(* CoDeSys 2.3.9.62 project: MM000-P9000-00-A.pro *)
(* Author: JvL *)
(* Libraries: ifm_RAWCan\ifm_RAWCan_NT_V020004.lib 1.10.19 08:10:40, ifm_CR0403\ifm_CR0403_V030100.lib 22.3.17 12:39:40, ifm_CANopen\ifm_NetVarLib_NT_V020004.lib 1.10.19 08:10:40, standard.lib 4.10.05 12:14:46, SysLibCallback.lib 26.9.08 18:43:52, 3S_CANOPENNETVAR.LIB 23.10.20 12:28:45, Iecsfc.lib 2.6.14 11:37:46, Util.lib 23.10.20 12:25:49, ifm_CANopen\3S_CANopenManager.lib 23.10.20 12:28:45, ifm_CANopen\3S_CanDrv.lib 23.10.20 12:28:45 *)

(* PLC configuration (modules and I/O channels)
Configuration [LocalConfiguration] node 0, in %IB0 out %QB0 {IFM_PARAM_WORD_TIME = 0}
Inputs Binary [LocalIn] node 0, in %IB0 out %QB0
  IN00 AT %IB0 [ChInputBool] Input 00 Bit
  IN01 AT %IB1 [ChInputBool] Input 01 Bit
  IN02 AT %IB2 [ChInputBool] Input 02 Bit
  IN03 AT %IB3 [ChInputBool] Input 03 Bit
  IN04 AT %IB4 [ChInputBool] Input 04 Bit
  IN05 AT %IB5 [ChInputBool] Input 05 Bit
  IN06 AT %IB6 [ChInputBool] Input 06 Bit
  IN07 AT %IB7 [ChInputBool] Input 07 Bit
  IN08 AT %IB8 [ChInputBool] Input 08 Bit
  IN09 AT %IB9 [ChInputBool] Input 09 Bit
  IN10 AT %IB10 [ChInputBool] Input 10 Bit
  IN11 AT %IB11 [ChInputBool] Input 11 Bit
Outputs Binary [LocalOut] node 1, in %IB12 out %QB0
  OUT00 AT %QB0 [ChOutputBool] Output 00 Bit
  OUT01 AT %QB1 [ChOutputBool] Output 01 Bit
  OUT02 AT %QB2 [ChOutputBool] Output 02 Bit
  OUT03 AT %QB3 [ChOutputBool] Output 03 Bit
  OUT04 AT %QB4 [ChOutputBool] Output 04 Bit
  OUT05 AT %QB5 [ChOutputBool] Output 05 Bit
  OUT06 AT %QB6 [ChOutputBool] Output 06 Bit
  OUT07 AT %QB7 [ChOutputBool] Output 07 Bit
  OUT08 AT %QB8 [ChOutputBool] Output 08 Bit
  OUT09 AT %QB9 [ChOutputBool] Output 09 Bit
  OUT10 AT %QB10 [ChOutputBool] Output 10 Bit
  OUT11 AT %QB11 [ChOutputBool] Output 11 Bit
SUPPLY_VOLTAGE_VBBS AT %IW6 [ChInputWord] Supply voltage VBBS
SUPPLY_VOLTAGE_VU AT %IW7 [ChInputWord] Supply voltage VU
SUPPLY_VOLTAGE_VBB1 AT %IW8 [ChInputWord] Supply voltage VBB1
SUPPLY_VOLTAGE_VBB2 AT %IW9 [ChInputWord] Supply voltage VBB2
TEMPERATURE AT %IW10 [ChInputInt] Temperature
CAN Communication [LocalCANCom] node 2, in %IB22 out %QB12
  Interface CAN 1 [CAN_BUS] node 0, in %IB22 out %QB12 {STACK_DWORD_S = 0}
    CANopen Interface [CAN_OPEN] node 0, in %IB22 out %QB12
    J1939 Interface [CAN_J1939] node 1, in %IB22 out %QB12
  Interface CAN 2 [CAN_BUS] node 1, in %IB22 out %QB12 {STACK_DWORD_S = 0}
    CANopen Interface [CAN_OPEN] node 0, in %IB22 out %QB12
    J1939 Interface [CAN_J1939] node 1, in %IB22 out %QB12
*)

(* Global variable list: CanOpen implicit Variables *)
VAR_GLOBAL CONSTANT
	MAX_CTRLINDEX : INT := -1;
END_VAR

(* Global variable list: Global_Variables *)
VAR_GLOBAL
	encoderStatic:BOOL;
END_VAR

(* Global variable list: Networkmanagement implicit Variables CAN *)
VAR_GLOBAL CONSTANT
	USE_NWVARS_CAN : BOOL := TRUE;
	MAX_NetVarItems_CAN	: INT := 31;
	MAX_NetVarPDO_Rx_CAN	: INT := 3;
	MAX_NetVarPDO_Tx_CAN	: INT := 7;
	MAX_NetVarOD_CAN		: INT := 0;
END_VAR
VAR_GLOBAL
	pNetVarItems_CAN		: ARRAY[0..MAX_NetVarItems_CAN] OF NetVarDataItem_CAN;
	pNetVarPDO_Rx_CAN		: ARRAY[0..MAX_NetVarPDO_Rx_CAN] OF NetVarPDO_Rx_CAN;
	pNetVarPDO_Tx_CAN		: ARRAY[0..MAX_NetVarPDO_Tx_CAN] OF NetVarPDO_Tx_CAN;
	pNetVarOD_CAN			: ARRAY[0..MAX_NetVarOD_CAN] OF NetVarOD_CAN;
END_VAR

(* Global variable list: PDM_PLC_COMUNICATION2 *)
VAR_GLOBAL

	(*
	 System variables for basic comunication. CANopen TX/RX PDO1, PDO2, PDO3 and PDO4
	or CANLayer2 TX/RX COB1, COB2, COB3 and COB4
	*)


(************************************From PDM to PLC**********************************************************)

	PRESENT_PAGE:WORD;					(*Preset page number from PDM to PLC*)
	PRESENT_MESSAGE:BYTE;					(*Preset message number from PDM to PLC*)
	PRESENT_MESSAGE_GROUP:BYTE;		(*Preset message group number from PDM to PLC*)
	F_KEYS:BYTE;								(*Funtion keys F1 to F8 from PDM to PLC*)
	C_KEYS:BYTE;								(*Control keys from PDM to PLC*)
	PRESENT_LEDVALUE_MAX:BYTE;			(*Preset LED valus max from PDM to PLC*)
	PRESENT_LEDVALUE_NIGHT:BYTE;		(*Preset LED value night from PDM to PLC*)

	PRESENT_BACKLIGHT:BYTE;				(*Preset backlight value from PDM to PLC*)
	HANDLE:WORD;								(*Handle for input value to PLC*)
	INPUT_VALUE:DWORD;						(*Input value to PLC*)
	LENGHT:BYTE;								(*Length for input value*)

	F_KEYS2:				BYTE;					(*Funtion keys F9 to F16 from PDM to PLC*)
	ToPlcPdo3ReserveByte1:BYTE;					(*Reserve PDO*)
	ToPlcPdo3ReserveByte2:BYTE;					(*Reserve PDO*)
	ToPlcPdo3ReserveByte3:BYTE;					(*Reserve PDO*)
	ToPlcPdo3ReserveByte4:BYTE;					(*Reserve PDO*)
	ToPlcPdo3ReserveByte5:BYTE;					(*Reserve PDO*)
	ToPlcPdo3ReserveByte6:BYTE;					(*Reserve PDO*)
	ToPlcPdo3ReserveByte7:BYTE;					(*Reserve PDO*)

	ToPlcPdo4ReserveByte0:BYTE;					(*Reserve PDO*)
	ToPlcPdo4ReserveByte1:BYTE;					(*Reserve PDO*)
	ToPlcPdo4ReserveByte2:BYTE;					(*Reserve PDO*)
	ToPlcPdo4ReserveByte3:BYTE;					(*Reserve PDO*)
	ToPlcPdo4ReserveByte4:BYTE;					(*Reserve PDO*)
	ToPlcPdo4ReserveByte5:BYTE;					(*Reserve PDO*)
	ToPlcPdo4ReserveByte6:BYTE;					(*Reserve PDO*)
	ToPlcPdo4ReserveByte7:BYTE;					(*Reserve PDO*)

(*^^^^^^^^^^^^^^^^^^^^^^^^^^^^^^^^^^^^^^^^^^^^^^^^^^^^^^^^^^^^^^^^^^^^^^^^^^^^^^^^^^^^^^^^^^^^^^^^^^^^^^^^^^^^^^^^^^^^^^^^^^^^^^^^^^^^^^^^^^*)

(*********************************************From PLC to PDM****************************************************************************)

	DESIRED_PAGE:WORD;						(*Desired page number from PLC to PDM*)
	DESIRED_MESSAGE:BYTE;					(*Desired message number from PLC to PDM*)
	DESIRED_MESSAGE_GROUP:BYTE;		(*Desired message group number from PLC to PDM*)
	LED_F_KEYS:BYTE;							(*LED Funtion keys F1 to F8 from PLC to PDM*)
	LED_C_KEYS:BYTE;							(*LED Control keys from PLC to PDM*)
	DESIRED_LEDVALUE_MAX:BYTE;			(*Desired LED valus max from PLC to PDM*)
	DESIRED_LEDVALUE_NIGHT:BYTE;		(*Desired LED value night from PLC to PDM*)

	DESIRED_BACKLIGHT:BYTE;				(*Desired backlight value from PLC to PDM*)
	HANDLE_BACK:WORD;						(*Handle for input value, write back from PLC*)
	INPUT_VALUE_BACK:DWORD;				(*Input value, write back from PLC*)
	LENGHT_BACK:BYTE;						(*Length for input value, write back from PLC*)

	LED_F_KEYS2		:BYTE;					(*LED Funtion keys F9 to F16 from PLC to PDM*)
	ToPdmPdo3ReserveByte1:BYTE;					(*Reserve PDO*)
	ToPdmPdo3ReserveByte2:BYTE;					(*Reserve PDO*)
	ToPdmPdo3ReserveByte3:BYTE;					(*Reserve PDO*)
	ToPdmPdo3ReserveByte4:BYTE;					(*Reserve PDO*)
	ToPdmPdo3ReserveByte5:BYTE;					(*Reserve PDO*)
	ToPdmPdo3ReserveByte6:BYTE;					(*Reserve PDO*)
	ToPdmPdo3ReserveByte7:BYTE;					(*Reserve PDO*)

	ToPdmPdo4ReserveByte0:BYTE;					(*Reserve PDO*)
	ToPdmPdo4ReserveByte1:BYTE;					(*Reserve PDO*)
	ToPdmPdo4ReserveByte2:BYTE;					(*Reserve PDO*)
	ToPdmPdo4ReserveByte3:BYTE;					(*Reserve PDO*)
	ToPdmPdo4ReserveByte4:BYTE;					(*Reserve PDO*)
	ToPdmPdo4ReserveByte5:BYTE;					(*Reserve PDO*)
	ToPdmPdo4ReserveByte6:BYTE;					(*Reserve PDO*)
	ToPdmPdo4ReserveByte7:BYTE;					(*Reserve PDO*)

(*^^^^^^^^^^^^^^^^^^^^^^^^^^^^^^^^^^^^^^^^^^^^^^^^^^^^^^^^^^^^^^^^^^^^^^^^^^^^^^^^^^^^^^^^^^^^^^^^^^^^^^^^^^^^^^^^^^^^^^^^^^^^^^^^^^^^^^^^^^*)

END_VAR

(* POU PLC_PRG, FBD *)
PROGRAM PLC_PRG
(*******************************************************************************************************************

			Template for CR0403 V03 - CAN layer 2 (2014)
			--------------------------------------------

	Wir möchten an dieser Stelle ausdrücklich darauf hinweisen, dass die eingestellten Beispiele
	nicht ungeprüft industriell eingesetzt werden dürfen. Das heißt, dass wir für die Funktionalität
	insbesondere an Maschinen und Anlagen keinerlei Garantie übernehmen. Das Beispiel ist
	ausschließlich für Testzwecke bei der Entwicklung neuer Maschinen und Anlagen vorgesehen
	und wurde dafür in Abstimmung mit Ihnen konstruiert und hergestellt. Insoweit handelt es sich
	nicht um ein (Software-) Produkt, das von europäischen Richtlinien erfasst wird. Die Konformität
	mit einschlägigen Richtlinien und Normen zur Erfüllung der gesetzlichen Anforderungen für das
	Inverkehrbringen werden erst mit der Verifizierung und Validierung im Rahmen Ihrer Entwicklung
	festgestellt. Ein Bereitstellen auf dem Markt zur Verwendung durch Endnutzer darf bis zu diesem
	Zeitpunkt nicht stattfinden. 
 
 	We would like to expressly point out that the examples made available must not be used for industrial
	purposes without checking. We assume no guarantee whatsoever for their functionality, particularly
	regarding machines and plants. The example is only intended for testing during the development of
	new machines and plants and has been designed and manufactured for this purpose in coordination
	with you.  Consequently, it is not a (software) product subject to European directives. Compliance with
	relevant directives and standards to meet legal requirements regarding the placing on the market will
	only be determined during the verification and validation in the context of your development. Until then,
	it must not be put onto the market for use by end users.

*******************************************************************************************************************)
VAR

	Init1: BOOL:=TRUE;
	CycleTime:DWORD;
	MaxCycleTime:DWORD;
	ResetMax:BOOL;

	Start_time: TIME;


	Var1: BOOL;
	Dumy: BOOL;
	Wert1: BYTE;
END_VAR
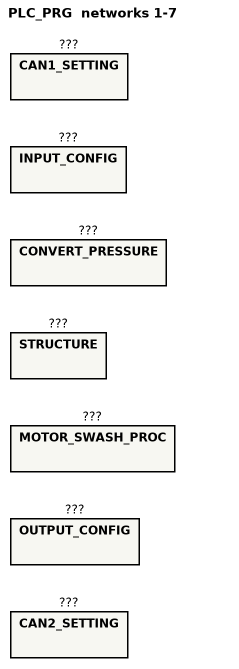
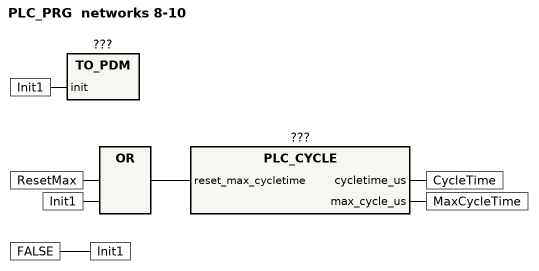
_FBD_ (* Function Block Diagram *)
NETWORK 1
	???:CAN1_SETTING()
NETWORK 2
	???:INPUT_CONFIG()
NETWORK 3
	???:CONVERT_PRESSURE()
NETWORK 4
	???:STRUCTURE()
NETWORK 5
	???:MOTOR_SWASH_PROC()
NETWORK 6
	???:OUTPUT_CONFIG()
NETWORK 7
	???:CAN2_SETTING()
NETWORK 8 (* If a PDM is not connected delete this line and the FB's TO_PDM and PLC_TO_PDM *)
	???:TO_PDM(init: Init1)
NETWORK 9
	???:PLC_CYCLE(reset_max_cycletime: OR(ResetMax, Init1), max_cycle_us => MaxCycleTime) => CycleTime
NETWORK 10 (* last line *)
	FALSE => Init1
_END_FBD_
(* the same logic as Structured Text *)
(* Network 1: see the listing above *)
(* Network 2: see the listing above *)
(* Network 3: see the listing above *)
(* Network 4: see the listing above *)
(* Network 5: see the listing above *)
(* Network 6: see the listing above *)
(* Network 7: see the listing above *)
(* Network 8: see the listing above *)
(* Network 9: see the listing above *)
(* Network 10 *)
Init1 := FALSE;
END_PROGRAM

(* POU CAN_SETTING/CAN1_SETTING, FBD *)
PROGRAM CAN1_SETTING
VAR
	CAN1_DownloadID: CAN_SETDOWNLOADID;
	CAN1_BaudRate: CAN_ENABLE;


	SetLed: SET_LED;
	LedFreq: BYTE:=2;
	Color1: BYTE := 2;
	Color2: BYTE := 0;
	ResultLed: BYTE;
	SettingsCAN: CAN_SETTING_ST;
END_VAR
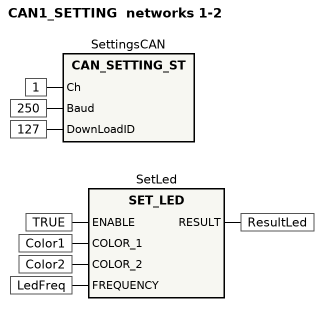
_FBD_ (* Function Block Diagram *)
NETWORK 1 (* Basic functions for the CAN / CANopen functionality *)
	SettingsCAN:CAN_SETTING_ST(Ch: 1, Baud: 250, DownLoadID: 127)
NETWORK 2
	SetLed:SET_LED(ENABLE: TRUE, COLOR_1: Color1, COLOR_2: Color2, FREQUENCY: LedFreq) => ResultLed
_END_FBD_
(* the same logic as Structured Text *)
(* Network 1: Basic functions for the CAN / CANopen functionality *)
SettingsCAN(Ch := 1, Baud := 250, DownLoadID := 127);
(* Network 2 *)
SetLed(ENABLE := TRUE, COLOR_1 := Color1, COLOR_2 := Color2, FREQUENCY := LedFreq);
ResultLed := SetLed.RESULT;
END_PROGRAM

(* POU CAN_SETTING/CAN_SETTING_ST, ST *)
FUNCTION_BLOCK CAN_SETTING_ST
(* Basic functions for the CAN / CANopen functionality *)
VAR

	CAN_SETDOWNLOADID_: CAN_SETDOWNLOADID;
	CAN_ENABLE_: CAN_ENABLE;

END_VAR
VAR_INPUT
	Ch: BYTE;
	Baud:WORD;
	DownLoadID:BYTE;
END_VAR
CAN_SETDOWNLOADID_(EXECUTE:=TRUE , CHANNEL:=Ch , DOWNLOAD_ID:=DownLoadID , RESULT=> );
CAN_ENABLE_(ENABLE:=TRUE , CHANNEL:=Ch , BAUDRATE:=Baud , RESULT=> );
END_FUNCTION_BLOCK

(* POU IO_CONFIGURATION/INPUT_CONFIG, FBD *)
PROGRAM INPUT_CONFIG
VAR
	fbEncoder: INC_ENCODER;
	TIMEBASE: TIME:=T#500ms;
	fbFrequency: PERIOD;
	result: BYTE;
	fbVoltage01: INPUT;
	fbInput01: INPUT;
END_VAR
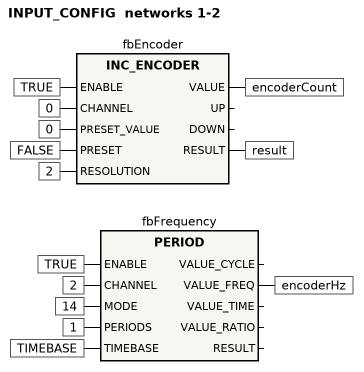
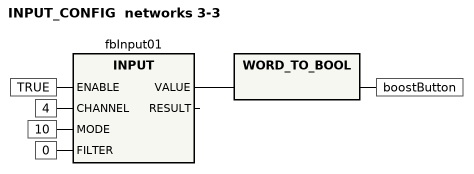
_FBD_ (* Function Block Diagram *)
NETWORK 1 (* This function block reads the encoder pulses and outputs a corresponding count value *)
	fbEncoder:INC_ENCODER(ENABLE: TRUE, CHANNEL: 0, PRESET_VALUE: 0, PRESET: FALSE, RESOLUTION: 2, RESULT => result) => encoderCount
NETWORK 2 (* This function block outputs the frequency of the encoder pulses in rpm *)
	fbFrequency:PERIOD(ENABLE: TRUE, CHANNEL: 2, MODE: 14, PERIODS: 1, TIMEBASE: TIMEBASE, VALUE_FREQ => encoderHz)
NETWORK 3
	WORD_TO_BOOL(fbInput01:INPUT(ENABLE: TRUE, CHANNEL: 4, MODE: 10, FILTER: 0)) => boostButton
_END_FBD_
(* the same logic as Structured Text *)
(* Network 1: This function block reads the encoder pulses and outputs a corresponding count value *)
fbEncoder(ENABLE := TRUE, CHANNEL := 0, PRESET_VALUE := 0, PRESET := FALSE, RESOLUTION := 2);
result := fbEncoder.RESULT;
encoderCount := fbEncoder.VALUE;
(* Network 2: This function block outputs the frequency of the encoder pulses in rpm *)
fbFrequency(ENABLE := TRUE, CHANNEL := 2, MODE := 14, PERIODS := 1, TIMEBASE := TIMEBASE);
encoderHz := fbFrequency.VALUE_FREQ;
(* Network 3 *)
fbInput01(ENABLE := TRUE, CHANNEL := 4, MODE := 10, FILTER := 0);
boostButton := WORD_TO_BOOL(fbInput01.VALUE);
END_PROGRAM

(* POU FUNCTIONAL_PROCEDURES/PDM_COM_LAYER2/CONVERT_PRESSURE, ST *)
PROGRAM CONVERT_PRESSURE
VAR
END_VAR
IF pressureRaw01 <= 4000 THEN
	motorWindinPsi := 0;
ELSIF pressureRaw01 >= 20000 THEN
	motorWindinPsi := 20000;
ELSE
	motorWindinPsi := REAL_TO_INT((pressureRaw01 - 4000) / 2.756);
END_IF

IF pressureRaw02 <= 4000 THEN
	motorPayoutPsi := 0;
ELSIF pressureRaw02 >= 20000 THEN
	motorPayoutPsi := 20000;
ELSE
	motorPayoutPsi := REAL_TO_INT((pressureRaw02 - 4000) / 2.756);
END_IF

IF pressureRaw03 <= 4000 THEN
	counterbalancePsi := 0;
ELSIF pressureRaw03 >= 20000 THEN
	counterbalancePsi := 20000;
ELSE
	counterbalancePsi := REAL_TO_INT((pressureRaw03 - 4000) / 2.756);
END_IF
END_PROGRAM

(* POU FUNCTIONAL_PROCEDURES/STRUCTURE, ST *)
PROGRAM STRUCTURE
VAR
	speedStatic:BOOL;
	motorSpeed: REAL;
	lastHighSpeedMode: BOOL;
	Delay: TON;
END_VAR
(* Reset software version number for new software versions*)
cr0403VersionNo := '000-00-A';
cr0431VersionNo := cr0431Version;

motorSpeed := (encoderHz * 60 * 34.20) / 500;

(*IF pressureRaw01 < 3500 OR pressureRaw02 < 3500 THEN
	sensorFailure:= TRUE;
	alarmBuzzer:= TRUE;
ELSE
	*)sensorFailure:= FALSE;(*
END_IF*)

IF waterBrake < 1000 OR bandBrake < 1000 THEN
	brakesOn:= TRUE;
ELSE
	brakesOn:= FALSE;
END_IF

IF encoderHz = 0 THEN
	speedStatic:= TRUE;
ELSE
	speedStatic:=FALSE;
END_IF

(* Boost mode functionality is activated when the boost button is pressed*)
IF boostButton AND motorSpeed > 500 THEN
	IF highSpeedMode <> lastHighSpeedMode THEN
		Delay(IN:=NOT(Delay.Q), PT:=T#1s);
		IF Delay.Q THEN
			CHANGE_DISPLACEMENT_PROC();
		END_IF
	ELSE
		CHANGE_DISPLACEMENT_PROC();
	END_IF
ELSE
	highSpeedMode := FALSE;
END_IF

(*IF encoderStatic <> speedStatic THEN
	sensorFailure:= TRUE;
	alarmBuzzer:=TRUE;
ELSE*)
	sensorFailure:=FALSE;
(*END_IF*)

joystick:=joystickPosition;
parkBrake:=applyParkbrake;
skylineClutch:=releaseSkylineClutch;

IF skylineActive = TRUE AND sensorFailure = FALSE THEN
	activateJoystick:= TRUE;
	IF joystickPosition >= 5100 THEN
		applyParkBrake:= FALSE;
		IF overloadWarning = FALSE THEN
			waterBrake:= 1000;
			bandBrake:= 1000;
			OVERLOAD_PROC();
		END_IF
	ELSIF joystickPosition <= 4900 THEN
		applyParkBrake:= FALSE;
		IF overspeedAlarm = FALSE THEN
			waterBrake:= 1000;
			bandBrake:= 1000;
		END_IF
		OVERSPEED_PROC();
	ELSE
		IF overloadWarning OR overspeedAlarm THEN
			Delay(IN:=NOT(Delay.Q), PT:=T#3s);
			IF Delay.Q THEN
				overloadWarning:= FALSE;
				overspeedAlarm:= FALSE;
			END_IF
		END_IF
		waterBrake:= 0;
		bandBrake:= 0;
		overspeedWarning:= FALSE;
		alarmBuzzer:= FALSE;
		IF encoderHz = 0 THEN
			applyParkBrake:= TRUE;
		END_IF
	END_IF
ELSIF sensorFailure = TRUE THEN
	alarmBuzzer:= TRUE;
ELSE
	activateJoystick:= FALSE;
	waterBrake:= 0;
	bandBrake:= 0;
	alarmBuzzer:= FALSE;
	IF encoderHz = 0 THEN
		applyParkBrake:= TRUE;
	END_IF
END_IF
END_PROGRAM

(* POU FUNCTIONAL_PROCEDURES/CHANGE_DISPLACEMENT_PROC, FBD *)
PROGRAM CHANGE_DISPLACEMENT_PROC
VAR
	fbHysteresis01: HYSTERESIS;
	value: INT;
END_VAR
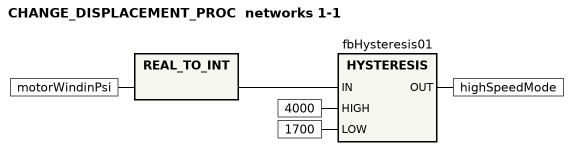
_FBD_ (* Function Block Diagram *)
NETWORK 1 (* This function block indicates when to change the motor to max displacement. / Goes TRUE if the pressure exceeds 4000psi and goes FALSE if the pressure falls back below 1700psi. *)
	fbHysteresis01:HYSTERESIS(IN: REAL_TO_INT(motorWindinPsi), HIGH: 4000, LOW: 1700) => highSpeedMode
_END_FBD_
(* the same logic as Structured Text *)
(* Network 1: This function block indicates when to change the motor to max displacement. / Goes TRUE if the pressure exceeds 4000psi and goes FALSE if the pressure falls back below 1700psi. *)
fbHysteresis01(IN := REAL_TO_INT(motorWindinPsi), HIGH := 4000, LOW := 1700);
highSpeedMode := fbHysteresis01.OUT;
END_PROGRAM

(* POU FUNCTIONAL_PROCEDURES/OVERLOAD_PROC, ST *)
PROGRAM OVERLOAD_PROC
VAR
	lastEncoderCount: DINT;
END_VAR
(* Check if drum is spinning in a payout direction *)

IF encoderCount > lastEncoderCount THEN
	waterBrake:= 0;
	overloadWarning:= TRUE;
	alarmBuzzer:= TRUE;
	encoderStatic:=FALSE;
ELSIF encoderCount = lastEncoderCount THEN
	encoderStatic:= TRUE;
ELSE
	encoderStatic:= FALSE;
END_IF

lastEncoderCount := encoderCount;
END_PROGRAM

(* POU FUNCTIONAL_PROCEDURES/OVERSPEED_PROC, ST *)
PROGRAM OVERSPEED_PROC
VAR
	motorSpeed: REAL;
END_VAR
(* This procedure checks the motor speed and signals the approriate action to prevent an overspeed event *)

motorSpeed := (encoderHz * 60 * 34.20) / 500; (*converting encoder Hz to actual motor speed in rpm, set encoder to 250 ppr=500 total pulses per rev*)
IF highSpeedMode THEN		(*Speed limits differ depending on motor speed setting*)
	IF motorSpeed > 4400 THEN
		waterBrake := 1000-(bandLimitSetpoint * 10);
		bandBrake := 1000-(bandLimitSetpoint * 10);
		releaseSkylineClutch := TRUE;
		overspeedWarning := FALSE;
		overspeedAlarm := TRUE;
		alarmBuzzer := TRUE;
	ELSIF motorSpeed > 3960 THEN
		waterBrake := 1000-(wcbLimitSetpoint * 10);
		bandBrake := 1000;
		releaseSkylineClutch := FALSE;
		overspeedWarning := FALSE;
		overspeedAlarm := TRUE;
		alarmBuzzer := TRUE;
	ELSIF motorSpeed > 3520 THEN
		waterBrake := 1000;
		bandBrake := 1000;
		releaseSkylineClutch := FALSE;
		overspeedWarning := TRUE;
		overspeedAlarm := FALSE;
		alarmBuzzer := FALSE;
	ELSE
		waterBrake := 1000;
		bandBrake := 1000;
		releaseSkylineClutch := FALSE;
		overspeedWarning := FALSE;
		overspeedAlarm := FALSE;
		alarmBuzzer := FALSE;
	END_IF
ELSE
	IF motorSpeed > 2780 THEN
		waterBrake := 1000-(bandLimitSetpoint * 10);
		bandBrake := 1000-(bandLimitSetpoint * 10);
		releaseSkylineClutch := TRUE;
		overspeedWarning := FALSE;
		overspeedAlarm := TRUE;
		alarmBuzzer := TRUE;
	ELSIF motorSpeed > 2500 THEN
		waterBrake := 1000-(wcbLimitSetpoint * 10);
		bandBrake := 1000;
		releaseSkylineClutch := FALSE;
		overspeedWarning := FALSE;
		overspeedAlarm := TRUE;
		alarmBuzzer := TRUE;
	ELSIF motorSpeed > 2230 THEN
		waterBrake :=1000;
		bandBrake := 1000;
		releaseSkylineClutch := FALSE;
		overspeedWarning := TRUE;
		overspeedAlarm := FALSE;
		alarmBuzzer := FALSE;
	ELSE
		waterBrake := 1000;
		bandBrake :=1000;
		releaseSkylineClutch := FALSE;
		overspeedWarning := FALSE;
		overspeedAlarm := FALSE;
		alarmBuzzer := FALSE;
	END_IF
END_IF
END_PROGRAM

(* POU FUNCTIONAL_PROCEDURES/MOTOR_SWASH_PROC, ST *)
PROGRAM MOTOR_SWASH_PROC
VAR
END_VAR
IF highSpeedMode THEN
	motorSwash:= 1000;
ELSE
	motorSwash:= 0;
END_IF
END_PROGRAM

(* POU IO_CONFIGURATION/OUTPUT_CONFIG, FBD *)
PROGRAM OUTPUT_CONFIG
VAR
	fbPwm01: PWM1000;
	fbPwm02: PWM1000;
	fbPwm03: PWM1000;
	fbBuzzer01: OUTPUT;
	fbBlink01: BLINK;
END_VAR
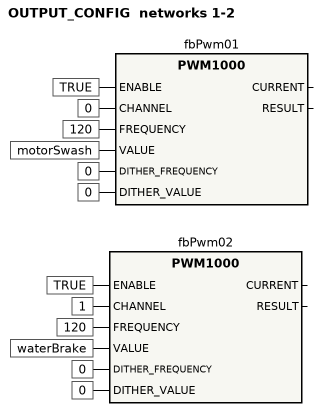
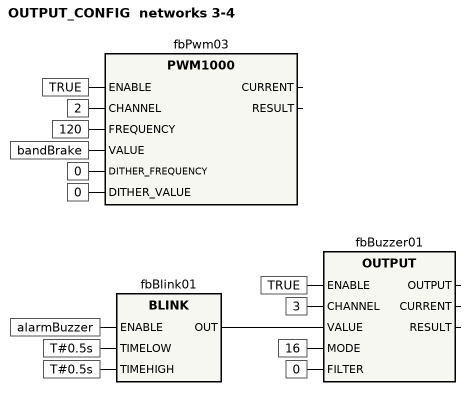
_FBD_ (* Function Block Diagram *)
NETWORK 1
	fbPwm01:PWM1000(ENABLE: TRUE, CHANNEL: 0, FREQUENCY: 120, VALUE: motorSwash, DITHER_FREQUENCY: 0, DITHER_VALUE: 0)
NETWORK 2
	fbPwm02:PWM1000(ENABLE: TRUE, CHANNEL: 1, FREQUENCY: 120, VALUE: waterBrake, DITHER_FREQUENCY: 0, DITHER_VALUE: 0)
NETWORK 3
	fbPwm03:PWM1000(ENABLE: TRUE, CHANNEL: 2, FREQUENCY: 120, VALUE: bandBrake, DITHER_FREQUENCY: 0, DITHER_VALUE: 0)
NETWORK 4 (* When alarmBuzzer is TRUE the buzzer will sound at a 1 Hz rate. *)
	fbBuzzer01:OUTPUT(ENABLE: TRUE, CHANNEL: 3, VALUE: fbBlink01:BLINK(ENABLE: alarmBuzzer, TIMELOW: T#0.5s, TIMEHIGH: T#0.5s), MODE: 16, FILTER: 0)
_END_FBD_
(* the same logic as Structured Text *)
(* Network 1 *)
fbPwm01(ENABLE := TRUE, CHANNEL := 0, FREQUENCY := 120, VALUE := motorSwash, DITHER_FREQUENCY := 0, DITHER_VALUE := 0);
(* Network 2 *)
fbPwm02(ENABLE := TRUE, CHANNEL := 1, FREQUENCY := 120, VALUE := waterBrake, DITHER_FREQUENCY := 0, DITHER_VALUE := 0);
(* Network 3 *)
fbPwm03(ENABLE := TRUE, CHANNEL := 2, FREQUENCY := 120, VALUE := bandBrake, DITHER_FREQUENCY := 0, DITHER_VALUE := 0);
(* Network 4: When alarmBuzzer is TRUE the buzzer will sound at a 1 Hz rate. *)
fbBlink01(ENABLE := alarmBuzzer, TIMELOW := T#0.5s, TIMEHIGH := T#0.5s);
fbBuzzer01(ENABLE := TRUE, CHANNEL := 3, VALUE := fbBlink01.OUT, MODE := 16, FILTER := 0);
END_PROGRAM

(* POU CAN_SETTING/CAN2_SETTING, FBD *)
PROGRAM CAN2_SETTING
VAR
	fbCan2: CAN_SETTING_ST;
END_VAR
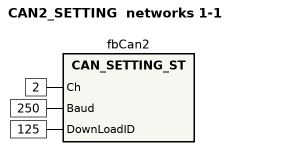
_FBD_ (* Function Block Diagram *)
NETWORK 1
	fbCan2:CAN_SETTING_ST(Ch: 2, Baud: 250, DownLoadID: 125)
_END_FBD_
(* the same logic as Structured Text *)
(* Network 1 *)
fbCan2(Ch := 2, Baud := 250, DownLoadID := 125);
END_PROGRAM

(* POU FUNCTIONAL_PROCEDURES/PDM_COM_LAYER2/TO_PDM, FBD *)
PROGRAM TO_PDM
VAR

	error_com: BOOL;
	led_f1: BOOL;
	led_f2: BOOL;
	led_f3: BOOL;
	led_f4: BOOL;
	led_f5: BOOL;
	led_f6: BOOL;
	led_esc: BOOL;
	led_up: BOOL;
	led_ok: BOOL;
	led_left: BOOL;
	led_down: BOOL;
	led_right: BOOL;


	F_key: UNPACK;
	F_key2: UNPACK;

	f1: BOOL;
	f2: BOOL;
	f3: BOOL;
	f4: BOOL;
	f5: BOOL;
	f6: BOOL;
	f7: BOOL;
	f8: BOOL;
	f9: BOOL;

	C_key: UNPACK;
	k_esc: BOOL;
	k_up: BOOL;
	k_ok: BOOL;
	k_left: BOOL;
	k_down: BOOL;
	k_right: BOOL;
	guard_time: TIME := T#500ms;

	led_f7: BOOL;
	led_f8: BOOL;
	led_f9: BOOL;
END_VAR
VAR_INPUT
	init: BOOL;
END_VAR
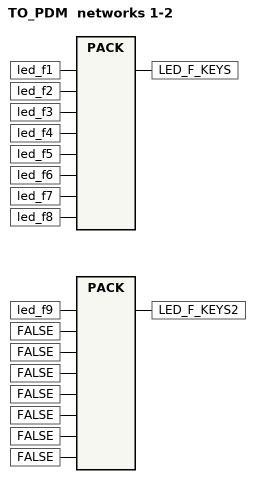
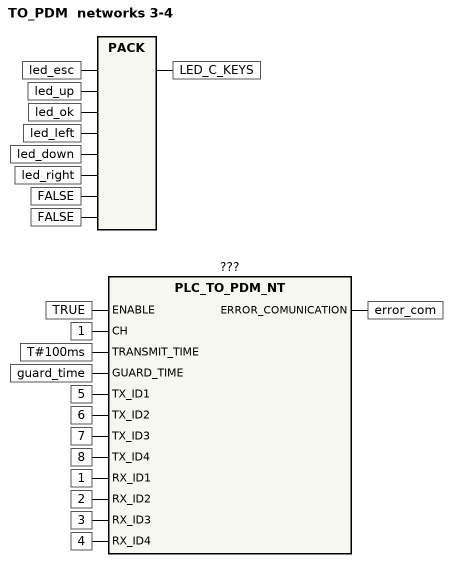
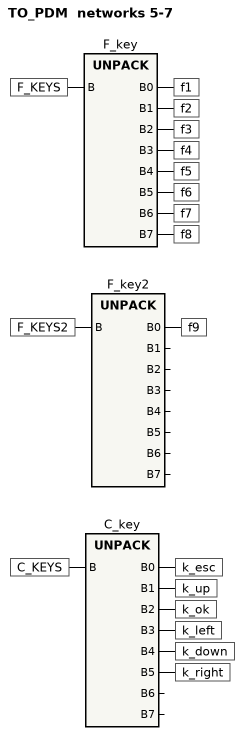
_FBD_ (* Function Block Diagram *)
NETWORK 1
	PACK(led_f1, led_f2, led_f3, led_f4, led_f5, led_f6, led_f7, led_f8) => LED_F_KEYS
NETWORK 2
	PACK(led_f9, FALSE, FALSE, FALSE, FALSE, FALSE, FALSE, FALSE) => LED_F_KEYS2
NETWORK 3
	PACK(led_esc, led_up, led_ok, led_left, led_down, led_right, FALSE, FALSE) => LED_C_KEYS
NETWORK 4
	???:PLC_TO_PDM_NT(ENABLE: TRUE, CH: 1, TRANSMIT_TIME: T#100ms, GUARD_TIME: guard_time, TX_ID1: 5, TX_ID2: 6, TX_ID3: 7, TX_ID4: 8, RX_ID1: 1, RX_ID2: 2, RX_ID3: 3, RX_ID4: 4) => error_com
NETWORK 5
	F_key:UNPACK(B: F_KEYS, B1 => f2, B2 => f3, B3 => f4, B4 => f5, B5 => f6, B6 => f7, B7 => f8) => f1
NETWORK 6
	F_key2:UNPACK(B: F_KEYS2) => f9
NETWORK 7
	C_key:UNPACK(B: C_KEYS, B1 => k_up, B2 => k_ok, B3 => k_left, B4 => k_down, B5 => k_right) => k_esc
_END_FBD_
(* the same logic as Structured Text *)
(* Network 1 *)
LED_F_KEYS := PACK(led_f1, led_f2, led_f3, led_f4, led_f5, led_f6, led_f7, led_f8);
(* Network 2 *)
LED_F_KEYS2 := PACK(led_f9, FALSE, FALSE, FALSE, FALSE, FALSE, FALSE, FALSE);
(* Network 3 *)
LED_C_KEYS := PACK(led_esc, led_up, led_ok, led_left, led_down, led_right, FALSE, FALSE);
(* Network 4: see the listing above *)
(* Network 5 *)
F_key(B := F_KEYS);
f2 := F_key.B1;
f3 := F_key.B2;
f4 := F_key.B3;
f5 := F_key.B4;
f6 := F_key.B5;
f7 := F_key.B6;
f8 := F_key.B7;
f1 := F_key.B0;
(* Network 6 *)
F_key2(B := F_KEYS2);
f9 := F_key2.B0;
(* Network 7 *)
C_key(B := C_KEYS);
k_up := C_key.B1;
k_ok := C_key.B2;
k_left := C_key.B3;
k_down := C_key.B4;
k_right := C_key.B5;
k_esc := C_key.B0;
END_PROGRAM

(* POU FUNCTIONAL_PROCEDURES/PDM_COM_LAYER2/PLC_TO_PDM_NT, ST *)
PROGRAM PLC_TO_PDM_NT
VAR_INPUT

	ENABLE: BOOL;
	CH: BYTE;
	TRANSMIT_TIME:TIME;	(*if transmit time=0, both id's transmit asynchron*)
	GUARD_TIME:TIME;
	TX_ID1: WORD;
	TX_ID2: WORD;
	TX_ID3: WORD;
	TX_ID4: WORD;
	RX_ID1:WORD;
	RX_ID2:WORD;
	RX_ID3:WORD;
	RX_ID4:WORD;


END_VAR
VAR_OUTPUT

	ERROR_COMUNICATION: BOOL;

END_VAR
VAR

	Send1: CAN_TX;
	Send2: CAN_TX;
	Send3: CAN_TX;
	Send4: CAN_TX;
	Rec1: CAN_RX;
	Rec2: CAN_RX;
	Rec3: CAN_RX;
	Rec4: CAN_RX;
	async_send1: BOOL;
	async_send2: BOOL;
	async_send3: BOOL;
	async_send4: BOOL;

	clock: BOOL;
	VarDword:DWORD;
	VarWord:WORD;
	T1: TON;
	one: BOOL;
	rec_ok: BOOL;

	Fl_rec_ok: R_TRIG;
	T_guard_on: TON;
	T_guard_off: TON;
	guard_clock_on: BOOL;
	guard_clock_off: BOOL;


	page_old: WORD;
	message_old: BYTE;
	message_group_old: BYTE;
	led_F_key_old: BYTE;
	led_control_key_old: BYTE;
	led_value_max_old: BYTE;
	led_value_night_old: BYTE;
	BacklightOld:BYTE;
	HandleOld:WORD;
	InputValueOld:DWORD;
	LengthOld:BYTE;



	NoGuarding: BOOL;

	LED_F_KEYS2Old: BYTE;
	ToPdmPdo3ReserveByte1Old: BYTE;
	ToPdmPdo3ReserveByte2Old: BYTE;
	ToPdmPdo3ReserveByte3Old: BYTE;
	ToPdmPdo3ReserveByte4Old: BYTE;
	ToPdmPdo3ReserveByte5Old: BYTE;
	ToPdmPdo3ReserveByte6Old: BYTE;
	ToPdmPdo3ReserveByte7Old: BYTE;
	ToPdmPdo4ReserveByte0Old: BYTE;
	ToPdmPdo4ReserveByte1Old: BYTE;
	ToPdmPdo4ReserveByte2Old: BYTE;
	ToPdmPdo4ReserveByte3Old: BYTE;
	ToPdmPdo4ReserveByte4Old: BYTE;
	ToPdmPdo4ReserveByte5Old: BYTE;
	ToPdmPdo4ReserveByte6Old: BYTE;
	ToPdmPdo4ReserveByte7Old: BYTE;


END_VAR
IF enable THEN
(****************Build a sync for transmit*************************)
	IF transmit_time<T#1ms THEN (*if no transmit time stop sync transmition*)
		NoGuarding:=TRUE;
		ELSE
			NoGuarding:=FALSE;
	END_IF;
	IF transmit_time< T#50ms THEN
		transmit_time:=T#50ms;
	END_IF;
	T1(IN:=NOT T1.Q , PT:=transmit_time );
	clock:= T1.Q;

(*^^^^^^^^^^^^^^^^^^^^^^^^^^^^^^^^^^^^^^^^^^^^^^^^^^^^^^^^^^^^^^^^^^*)
(*************************Build the async for transmit*****************)
	IF page_old<>DESIRED_PAGE THEN
		page_old:=DESIRED_PAGE;
		async_send1:=TRUE;
	END_IF;
	IF message_old<>DESIRED_MESSAGE THEN
		message_old:=DESIRED_MESSAGE;
		async_send1:=TRUE;
	END_IF;
	IF message_group_old<>DESIRED_MESSAGE_GROUP THEN
		message_group_old:=DESIRED_MESSAGE_GROUP;
		async_send1:=TRUE;
	END_IF;
	IF led_F_key_old<>LED_F_KEYS THEN
		led_F_key_old:=LED_F_KEYS;
		async_send1:=TRUE;
	END_IF;
	IF led_control_key_old<>LED_C_KEYS THEN
		led_control_key_old:=LED_C_KEYS;
		async_send1:=TRUE;
	END_IF;
	IF led_value_max_old<>DESIRED_LEDVALUE_MAX THEN
		led_value_max_old:=DESIRED_LEDVALUE_MAX;
		async_send1:=TRUE;
	END_IF;
	IF led_value_night_old<>DESIRED_LEDVALUE_NIGHT THEN
		led_value_night_old:=DESIRED_LEDVALUE_NIGHT;
		async_send1:=TRUE;
	END_IF;
	IF DESIRED_BACKLIGHT>100 THEN
		DESIRED_BACKLIGHT:=100;
	END_IF;
	IF BacklightOld<>DESIRED_BACKLIGHT THEN
		BacklightOld:=DESIRED_BACKLIGHT;
		async_send2:=TRUE;
	END_IF;
	IF HandleOld<>HANDLE_BACK THEN
		HandleOld:=HANDLE_BACK;
		async_send2:=TRUE;
	END_IF;
	IF InputValueOld<>INPUT_VALUE_BACK THEN
		InputValueOld:=INPUT_VALUE_BACK;
		async_send2:=TRUE;
	END_IF;
	IF LengthOld<>LENGHT_BACK THEN
		LengthOld:=LENGHT_BACK;
		async_send2:=TRUE;
	END_IF;

	IF LED_F_KEYS2Old<>LED_F_KEYS2 THEN
		LED_F_KEYS2Old:=LED_F_KEYS2;
		async_send3:=TRUE;
	END_IF;
	IF ToPdmPdo3ReserveByte1Old<>ToPdmPdo3ReserveByte1 THEN
		ToPdmPdo3ReserveByte1Old:=ToPdmPdo3ReserveByte1;
		async_send3:=TRUE;
	END_IF;
	IF ToPdmPdo3ReserveByte2Old<>ToPdmPdo3ReserveByte2 THEN
		ToPdmPdo3ReserveByte2Old:=ToPdmPdo3ReserveByte2;
		async_send3:=TRUE;
	END_IF;
	IF ToPdmPdo3ReserveByte3Old<>ToPdmPdo3ReserveByte3 THEN
		ToPdmPdo3ReserveByte3Old:=ToPdmPdo3ReserveByte3;
		async_send3:=TRUE;
	END_IF;
	IF ToPdmPdo3ReserveByte4Old<>ToPdmPdo3ReserveByte4 THEN
		ToPdmPdo3ReserveByte4Old:=ToPdmPdo3ReserveByte4;
		async_send3:=TRUE;
	END_IF;
	IF ToPdmPdo3ReserveByte5Old<>ToPdmPdo3ReserveByte5 THEN
		ToPdmPdo3ReserveByte5Old:=ToPdmPdo3ReserveByte5;
		async_send3:=TRUE;
	END_IF;
	IF ToPdmPdo3ReserveByte6Old<>ToPdmPdo3ReserveByte6 THEN
		ToPdmPdo3ReserveByte6Old:=ToPdmPdo3ReserveByte6;
		async_send3:=TRUE;
	END_IF;
	IF ToPdmPdo3ReserveByte7Old<>ToPdmPdo3ReserveByte7 THEN
		ToPdmPdo3ReserveByte7Old:=ToPdmPdo3ReserveByte7;
		async_send3:=TRUE;
	END_IF;
	IF ToPdmPdo4ReserveByte0Old<>ToPdmPdo4ReserveByte0 THEN
		ToPdmPdo4ReserveByte0Old:=ToPdmPdo4ReserveByte0;
		async_send4:=TRUE;
	END_IF;
	IF ToPdmPdo4ReserveByte1Old<>ToPdmPdo4ReserveByte1 THEN
		ToPdmPdo4ReserveByte1Old:=ToPdmPdo4ReserveByte1;
		async_send4:=TRUE;
	END_IF;
	IF ToPdmPdo4ReserveByte2Old<>ToPdmPdo4ReserveByte2 THEN
		ToPdmPdo4ReserveByte2Old:=ToPdmPdo4ReserveByte2;
		async_send4:=TRUE;
	END_IF;
	IF ToPdmPdo4ReserveByte3Old<>ToPdmPdo4ReserveByte3 THEN
		ToPdmPdo4ReserveByte3Old:=ToPdmPdo4ReserveByte3;
		async_send4:=TRUE;
	END_IF;
	IF ToPdmPdo4ReserveByte4Old<>ToPdmPdo4ReserveByte4 THEN
		ToPdmPdo4ReserveByte4Old:=ToPdmPdo4ReserveByte4;
		async_send4:=TRUE;
	END_IF;
	IF ToPdmPdo4ReserveByte5Old<>ToPdmPdo4ReserveByte5 THEN
		ToPdmPdo4ReserveByte5Old:=ToPdmPdo4ReserveByte5;
		async_send4:=TRUE;
	END_IF;
	IF ToPdmPdo4ReserveByte6Old<>ToPdmPdo4ReserveByte6 THEN
		ToPdmPdo4ReserveByte6Old:=ToPdmPdo4ReserveByte6;
		async_send4:=TRUE;
	END_IF;
	IF ToPdmPdo4ReserveByte7Old<>ToPdmPdo4ReserveByte7 THEN
		ToPdmPdo4ReserveByte7Old:=ToPdmPdo4ReserveByte7;
		async_send4:=TRUE;
	END_IF;



(*^^^^^^^^^^^^^^^^^^^^^^^^^^^^^^^^^^^^^^^^^^^^^^^^^^^^^^^^^^^^^^^^^^*)

(************Build the guarding toggle and send it with backlight*****************************)

	IF clock THEN
		one := NOT one;
	END_IF;

	Send2.DATA[0]:=DESIRED_BACKLIGHT;

	IF one THEN
		Send2.DATA[0].7:= TRUE;
		ELSE
			Send2.DATA[0].7:=FALSE;
	END_IF;
(*^^^^^^^^^^^^^^^^^^^^^^^^^^^^^^^^^^^^^^^^^^^^^^^^^^^^^^^^^^^^^^^^^^*)

(********************copy data to transmit array*********************)

	Send1.DATA[0] := WORD_TO_BYTE(DESIRED_PAGE);
	VarWord := SHR(DESIRED_PAGE,8);
	Send1.DATA[1] := WORD_TO_BYTE(VarWord);
	Send1.DATA[2] := DESIRED_MESSAGE;
	Send1.DATA[3] := DESIRED_MESSAGE_GROUP;
	Send1.DATA[4] := LED_F_KEYS;
	Send1.DATA[5] := LED_C_KEYS;
	Send1.DATA[6] := DESIRED_LEDVALUE_MAX;
	Send1.DATA[7] := DESIRED_LEDVALUE_NIGHT;

	IF LENGHT_BACK<1 THEN
		LENGHT_BACK:=1;
	END_IF;
	IF LENGHT_BACK=3 OR LENGHT_BACK>4 THEN
		LENGHT_BACK:=4;
	END_IF;

	Send2.DATA[7]:=LENGHT_BACK;

	Send2.DATA[1] := WORD_TO_BYTE(HANDLE_BACK);
	VarWord := SHR(HANDLE_BACK,8);
	Send2.DATA[2] := WORD_TO_BYTE(VarWord);


	CASE LENGHT_BACK OF

		1:	Send2.DATA[3]:=DWORD_TO_BYTE(INPUT_VALUE_BACK);
			Send2.DATA[4]:=0;
			Send2.DATA[5]:=0;
			Send2.DATA[6]:=0;

		2:	VarDword:=ROL(INPUT_VALUE_BACK,32);
			Send2.DATA[3]:=DWORD_TO_BYTE(VarDword);
			VarDword:=ROL(INPUT_VALUE_BACK,24);
			Send2.DATA[4]:=DWORD_TO_BYTE(VarDword);
			VarDword:=ROL(INPUT_VALUE_BACK,16);
			Send2.DATA[5]:=0;
			Send2.DATA[6]:=0;

		4:	VarDword:=ROL(INPUT_VALUE_BACK,32);
			Send2.DATA[3]:=DWORD_TO_BYTE(VarDword);
			VarDword:=ROL(INPUT_VALUE_BACK,24);
			Send2.DATA[4]:=DWORD_TO_BYTE(VarDword);
			VarDword:=ROL(INPUT_VALUE_BACK,16);
			Send2.DATA[5]:=DWORD_TO_BYTE(VarDword);
			VarDword:=ROL(INPUT_VALUE_BACK,8);
			Send2.DATA[6]:=DWORD_TO_BYTE(VarDword);

	END_CASE;

	Send3.DATA[0] := LED_F_KEYS2;
	Send3.DATA[1] := ToPdmPdo3ReserveByte1;
	Send3.DATA[2] := ToPdmPdo3ReserveByte2;
	Send3.DATA[3] := ToPdmPdo3ReserveByte3;
	Send3.DATA[4] := ToPdmPdo3ReserveByte4;
	Send3.DATA[5] := ToPdmPdo3ReserveByte5;
	Send3.DATA[6] := ToPdmPdo3ReserveByte6;
	Send3.DATA[7] := ToPdmPdo3ReserveByte7;

	Send4.DATA[0] := ToPdmPdo4ReserveByte0;
	Send4.DATA[1] := ToPdmPdo4ReserveByte1;
	Send4.DATA[2] := ToPdmPdo4ReserveByte2;
	Send4.DATA[3] := ToPdmPdo4ReserveByte3;
	Send4.DATA[4] := ToPdmPdo4ReserveByte4;
	Send4.DATA[5] := ToPdmPdo4ReserveByte5;
	Send4.DATA[6] := ToPdmPdo4ReserveByte6;
	Send4.DATA[7] := ToPdmPdo4ReserveByte7;


(*^^^^^^^^^^^^^^^^^^^^^^^^^^^^^^^^^^^^^^^^^^^^^^^^^^^^^^^^^^^^^^^^^^^^^^^^^^^^^^^^^^^^*)

(**************send data************************)
	Send1(
	ENABLE:=(clock AND NOT NoGuarding) OR async_send1 ,
	CHANNEL:=CH ,
	ID:=tx_id1 ,
	DATA:= ,
	RESULT=> );

	Send2(
	ENABLE:=(clock AND NOT NoGuarding) OR async_send2 ,
	CHANNEL:=CH ,
	ID:=tx_id2 ,
	DATA:= ,
	RESULT=> );

	Send3(
	ENABLE:=(clock AND NOT NoGuarding) OR async_send3 ,
	CHANNEL:=CH ,
	ID:=tx_id3 ,
	DATA:= ,
	RESULT=> );

	Send4(
	ENABLE:=(clock AND NOT NoGuarding) OR async_send4 ,
	CHANNEL:=CH ,
	ID:=tx_id4 ,
	DATA:= ,
	RESULT=> );

	async_send1:=FALSE;
	async_send2:=FALSE;
	async_send3:=FALSE;
	async_send4:=FALSE;


(*^^^^^^^^^^^^^^^^^^^^^^^^^^^^^^^^^^^^^^^^^^^^^^^^^^^^^^^^^^^^^^^^^^^^^^^^^^^^^^^^^^^^*)

(**************receive data************************)

	Rec1(
	ENABLE:=TRUE ,
	CHANNEL:=CH ,
	ID:=Rx_id1 ,
	DATA=> ,
	RESULT=> );

	Rec2(
	ENABLE:=TRUE ,
	CHANNEL:=CH ,
	ID:=Rx_id2 ,
	DATA=> ,
	RESULT=> );

	Rec3(
	ENABLE:=TRUE ,
	CHANNEL:=CH ,
	ID:=Rx_id3 ,
	DATA=> ,
	RESULT=> );

	Rec4(
	ENABLE:=TRUE ,
	CHANNEL:=CH ,
	ID:=Rx_id4 ,
	DATA=> ,
	RESULT=> );

	(**************************check guarding**********************************)
	Fl_rec_ok(CLK:=Rec2.DATA[0].7 , Q=>rec_ok );

	T_guard_on(IN:=rec_ok , PT:=guard_time , Q=>guard_clock_on);
	T_guard_off(IN:=NOT rec_ok , PT:=guard_time , Q=>guard_clock_off);


	IF NOT NoGuarding AND (guard_clock_on OR guard_clock_off) THEN
		error_comunication := TRUE;
		ELSE
			error_comunication := FALSE;
	END_IF;
	(*^^^^^^^^^^^^^^^^^^^^^^^^^^^^^^^^^^^^^^^^^^^^^^^^^^^^^^^^^^^^^^^^^^^^^^^^^^^^*)

	(***********************copy reveived data***********************************)
	IF Rec1.RESULT=1 THEN
		PRESENT_PAGE := Rec1.DATA[1];
		PRESENT_PAGE := SHL(PRESENT_PAGE,8) OR Rec1.DATA[0];
		PRESENT_MESSAGE := Rec1.DATA[2];
		PRESENT_MESSAGE_GROUP := Rec1.DATA[3];
		F_KEYS := Rec1.DATA[4];
		C_KEYS := Rec1.DATA[5];
		PRESENT_LEDVALUE_MAX := Rec1.DATA[6];
		PRESENT_LEDVALUE_NIGHT := Rec1.DATA[7];
	END_IF;

	IF Rec2.RESULT=1 THEN
		PRESENT_BACKLIGHT:= 16#7F AND Rec2.DATA[0];
		HANDLE:= BYTE_TO_WORD(Rec2.DATA[2]);
		HANDLE:=SHL(HANDLE,8);
		HANDLE:=HANDLE OR Rec2.DATA[1];
		LENGHT:= Rec2.DATA[7];

		IF LENGHT<1 THEN
			LENGHT:=1;
		END_IF;
		IF LENGHT=3 OR LENGHT>4 THEN
			LENGHT:=4;
		END_IF;
		CASE LENGHT OF
			1:	INPUT_VALUE:=Rec2.DATA[3];

			2:	INPUT_VALUE:=Rec2.DATA[4];
				INPUT_VALUE:=SHL(INPUT_VALUE,8) OR Rec2.DATA[3];

			4:	INPUT_VALUE:=Rec2.DATA[6];
				INPUT_VALUE:=SHL(INPUT_VALUE,8) OR Rec2.DATA[5];
				INPUT_VALUE:=SHL(INPUT_VALUE,8) OR Rec2.DATA[4];
				INPUT_VALUE:=SHL(INPUT_VALUE,8) OR Rec2.DATA[3];

		END_CASE;
	END_IF;

	IF Rec3.RESULT=1 THEN
		F_KEYS2:=Rec3.DATA[0];
		ToPlcPdo3ReserveByte1:=Rec3.DATA[1];
		ToPlcPdo3ReserveByte2:=Rec3.DATA[2];
		ToPlcPdo3ReserveByte3:=Rec3.DATA[3];
		ToPlcPdo3ReserveByte4:=Rec3.DATA[4];
		ToPlcPdo3ReserveByte5:=Rec3.DATA[5];
		ToPlcPdo3ReserveByte6:=Rec3.DATA[6];
		ToPlcPdo3ReserveByte7:=Rec3.DATA[7];
	END_IF;

	IF Rec4.RESULT=1 THEN
		ToPlcPdo4ReserveByte0:=Rec4.DATA[0];
		ToPlcPdo4ReserveByte1:=Rec4.DATA[1];
		ToPlcPdo4ReserveByte2:=Rec4.DATA[2];
		ToPlcPdo4ReserveByte3:=Rec4.DATA[3];
		ToPlcPdo4ReserveByte4:=Rec4.DATA[4];
		ToPlcPdo4ReserveByte5:=Rec4.DATA[5];
		ToPlcPdo4ReserveByte6:=Rec4.DATA[6];
		ToPlcPdo4ReserveByte7:=Rec4.DATA[7];
	END_IF;

	(*^^^^^^^^^^^^^^^^^^^^^^^^^^^^^^^^^^^^^^^^^^^^^^^^^^^^^^^^^^^^^^^^^^^^^^^^^^^^*)

(*^^^^^^^^^^^^^^^^^^^^^^^^^^^^^^^^^^^^^^^^^^^^^^^^^^^^^^^^^^^^^^^^^^^^^^^^^^^^^^^^^^^^^^^^^^^^^^^^^^^^^^^^^^^^^^^^^^^^^^^^^^^^^^^^^^^^^^^^^^^^*)
END_IF;
END_PROGRAM

(* POU PLC_CYCLE, ST *)
PROGRAM PLC_CYCLE
VAR
	old_cycle: DWORD;
	TIMER_READ_US1: TIMER_READ_US;
	cycle: DWORD;
	init: BOOL:=TRUE;
END_VAR
VAR_OUTPUT
	cycletime_us: DWORD;
	max_cycle_us: DWORD;
END_VAR

VAR_INPUT
	reset_max_cycletime: BOOL;
END_VAR
	TIMER_READ_US1(TIME_US=>cycle );
	cycletime_us:=cycle-old_cycle;
	old_cycle:=cycle;

	IF max_cycle_us<cycletime_us AND NOT init THEN
		max_cycle_us:=cycletime_us;
	END_IF;

	IF reset_max_cycletime THEN
		max_cycle_us:=0;
	END_IF;

	init:=FALSE;
END_PROGRAM
